(* CODESYS project dint.data.save.190523.1.project

Project tree, tasks and I/O mapping:
  MIC7001 : Changsha Xiangji-ARM Cortex A9(xilinx zynq7000)-linux, Changsha Xiangji Hiden Technology Co.Ltd, version 3.5.10.40
    application Application
      libraries: Standard, * (System); CAA File, * (CAA Technical Workgroup); CAA Types Extern, * (CAA Technical Workgroup); CAA Callback Extern, * (CAA Technical Workgroup); SysMem, * (System); Util, 3.5.11.0 (System); SysFile, 3.5.9.0 (System); SysTypes Interfaces, * (System); CAN API, 1.0.0.3 (3S - Smart Software Solutions GmbH); AC_DataLog, 3.5.12.0 (3S - Smart Software Solutions GmbH); SysTime, * (System); CAA DTUtil Extern, 3.5.12.0 (CAA Technical Workgroup); CAA SerialCom, 3.5.12.0 (CAA Technical Workgroup); cyber gpio, 3.5.10.40 (cyber)
      task MainTask (cyclic, interval 20 ms, priority 15) calls prg_dint_data_save
      trace Trace (task MainTask): g_ai_curr_prop_trace, g_ai_pilot_trace, g_ai_press_pump1_trace, g_ai_press_pump2_trace, GVL.g_rpm_trace
      program prg_dint_data_save [ST]
      function fn_write_dint_data [ST]
    SoftMotion General Axis Pool
  text list GlobalTextList
*)

// MIC7001/Application/prg_dint_data_save
PROGRAM prg_dint_data_save
VAR
	
	hFile: RTS_IEC_HANDLE := RTS_INVALID_HANDLE;
	
	i:UINT;
	curr_time : DWORD;
	pr:RTS_IEC_RESULT;
END_VAR

VAR_INPUT
	//可以在其它程序中修改本数组的值，在本程序中周期性保存
	save_data:ARRAY[0 .. 31] OF DINT;
	data_len:UINT := 12;  //需要与实际保存的数量一致
	
	//下面的变量为 True时，自动保存，为False，停止保存
	f_data_save:BOOL := FALSE;  
END_VAR


//保存实时数据. 每次以尾部添加方式写入原有数据文件，未考虑硬盘写满的处理，建议仅在主机开发调试阶段使用。

IF f_data_save = FALSE THEN   //停止写数据，关闭文件
	IF hFile <> RTS_INVALID_HANDLE THEN
		hFile := fn_write_dint_data(close := TRUE, num := data_len, hFile := hFile, pData := ADR(save_data));
		hFile := RTS_INVALID_HANDLE;
	END_IF
ELSE
	curr_time := SysTimeRtc.SysTimeRtcGet(pResult :=pr);
	save_data[0] := ANY_TO_DINT(curr_time); //保存时间

	hFile := fn_write_dint_data(close := FALSE, num := data_len, hFile := hFile, pData := ADR(save_data));
END_IF

END_PROGRAM

// MIC7001/Application/fn_write_dint_data
FUNCTION fn_write_dint_data : RTS_IEC_HANDLE
VAR_INPUT
	pData: POINTER TO DINT := 0;
	num:UINT := 0;	
	close:BOOL:= FALSE;
	hFile: RTS_IEC_HANDLE := RTS_INVALID_HANDLE;
END_VAR

VAR
	udiDeleteError: RTS_IEC_RESULT;
	udiOpenError: RTS_IEC_RESULT;
	udiWriteError: RTS_IEC_RESULT;
	udiSizeError: RTS_IEC_RESULT;
	filesize: __XWORD;
	i :DWORD;
	iTemp: UDINT;
	udiPos: UDINT;
	str: STRING(256);
	str_size: __XWORD;
	udiByteWrite: LWORD;
	check_sum:REAL := 0;
	gRandomNum :LWORD := 1;   //系统随机数,每个周期乘以内部传感器的实时值；
	filename:STRING := 'running_data_dint.txt';
END_VAR

fn_write_dint_data := RTS_INVALID_HANDLE;

IF close THEN
	IF hFile <> RTS_INVALID_HANDLE THEN
		sysfileclose(hFile := hFile);
		hFile := RTS_INVALID_HANDLE;
	END_IF
	fn_write_dint_data := RTS_INVALID_HANDLE;
	RETURN;
END_IF

IF hFile = RTS_INVALID_HANDLE THEN
	hFile := sysfileopen(szFile := filename, am := sysfile.AM_APPEND_PLUS, pResult:= ADR(udiOpenError));
	IF hFile = RTS_INVALID_HANDLE	THEN  //打开文件失败
		RETURN;
	END_IF
END_IF

filesize := sysfilegetsize(filename, ADR(udiSizeError));
udiPos := SysFileSetPos(hFile:=hFile, ulOffset:=filesize);	

str:= '';
FOR i := 0 TO num-1 DO
	str := concat(str, DINT_TO_STRING(pData[i]));
	str := concat(str, ',');
END_FOR

str := concat(str, '$N');		
str_size := ANY_TO_DWORD(len(str));

udiByteWrite := sysfile.SysFileWrite(hFile := hFile,pbyBuffer := ADR(str),ulSize := str_size, pResult := ADR(udiWriteError));

fn_write_dint_data := hFile;   //保持打开状态，下次继续写入

END_FUNCTION
